FUNCTION_BLOCK PauseSwitch (* Basic Function Block Type *)
  (* Standard: 61499-2 *)
  (* Version 0.0, 4/12/2016, Aalto_IT, nxtControl GmbH, Template *)
  PACKAGE Main;
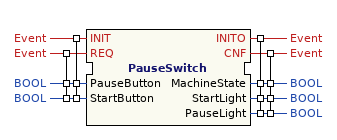
  EVENT_INPUT
    INIT WITH PauseButton, StartButton; (* Initialization Request *)
    REQ WITH PauseButton, StartButton; (* Normal Execution Request *)
  END_EVENT
  EVENT_OUTPUT
    INITO WITH MachineState, StartLight, PauseLight; (* Initialization Confirm *)
    CNF WITH MachineState, StartLight, PauseLight; (* Execution Confirmation *)
  END_EVENT
  VAR_INPUT
    PauseButton : BOOL; (* Input event qualifier *)
    StartButton : BOOL;
  END_VAR
  VAR_OUTPUT
    MachineState : BOOL; (* Output event qualifier *)
    StartLight : BOOL;
    PauseLight : BOOL;
  END_VAR
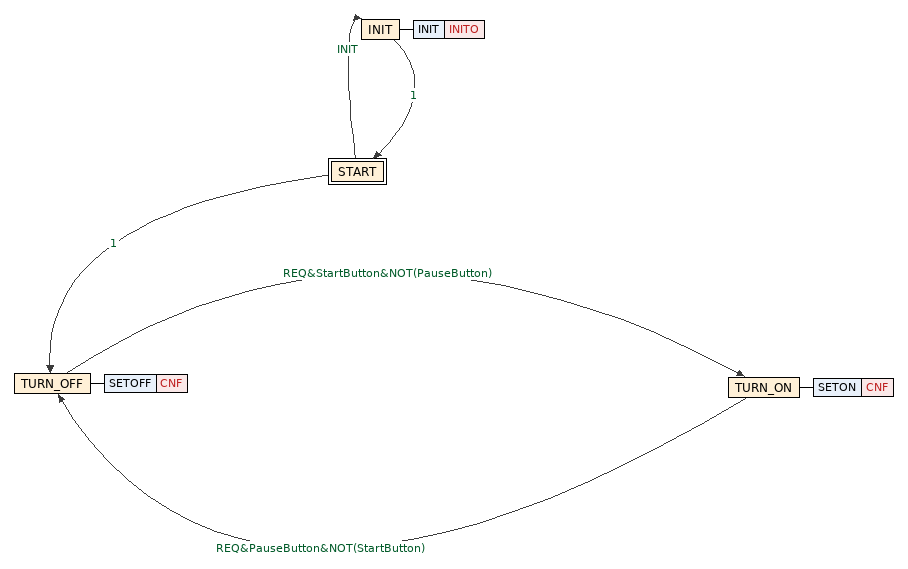
  EC_STATES
    START; (* Initial State *)
    INIT : INIT -> INITO; (* Initialization *)
    TURN_ON : SETON -> CNF; (* Normal execution *)
    TURN_OFF : SETOFF -> CNF; (* Normal execution *)
  END_STATES
  EC_TRANSITIONS
    START TO INIT := INIT;
    INIT TO START := 1;
    START TO TURN_OFF := 1;
    TURN_ON TO TURN_OFF := REQ&PauseButton&NOT(StartButton);
    TURN_OFF TO TURN_ON := REQ&StartButton&NOT(PauseButton);
  END_TRANSITIONS
  ALGORITHM INIT IN ST: (* Initialization algorithm *)
;
  END_ALGORITHM
  ALGORITHM SETON IN ST: (* Normally executed algorithm *)
;
MachineState:=1;
StartLight:=1;
PauseLight:=0;
  END_ALGORITHM
  ALGORITHM SETOFF IN ST:
;
MachineState:=0;
StartLight:=0;
PauseLight:=1;
  END_ALGORITHM
END_FUNCTION_BLOCK
